Fanuc KAREL source: kt00296.KL

-- PROVISIONAL review KL for V770-1; original PC SHA256 7c35b233e68bd5a4315989521f3a128318261ea5af6346b3853a4f87b088b54c
-- Incomplete behavior may be omitted. Consult companion uncertainty JSON. Do not deploy.
PROGRAM KT00296
%NOLOCKGROUP
VAR
  I1 : INTEGER
  OUT : BOOLEAN
-- UNRESOLVED_DECL H2 type=002017
BEGIN
  -- UNRESOLVED_PC offsets 5-16; opcodes 2E,23
  -- UNRESOLVED_PC offsets 21-35; opcodes 2E,22,9D,33,B4
  -- UNRESOLVED_PC offsets 40-62; opcodes 21,22,9D,33,B3,58,23
  -- UNRESOLVED_PC offsets 67-71; opcodes 7F
END KT00296
